FUNCTION_BLOCK numeroDePartidas (* Basic Function Block Type *)
  (* Standard: 61499-2 *)
  (* Version 0.0, 14/01/2026, Schneider Electric, Template *)
  PACKAGE Hidryco.HidrycoLib;
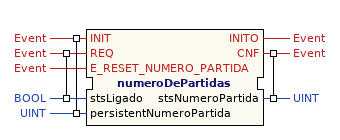
  EVENT_INPUT
    INIT WITH persistentNumeroPartida; (* Initialization Request *)
    REQ WITH stsLigado; (* Normal Execution Request *)
    E_RESET_NUMERO_PARTIDA;
  END_EVENT
  EVENT_OUTPUT
    INITO; (* Initialization Confirm *)
    CNF WITH stsNumeroPartida; (* Execution Confirmation *)
  END_EVENT
  VAR_INPUT
    stsLigado : BOOL;
    persistentNumeroPartida : UINT;
  END_VAR
  VAR_OUTPUT
    stsNumeroPartida : UINT; (* Output event qualifier *)
  END_VAR
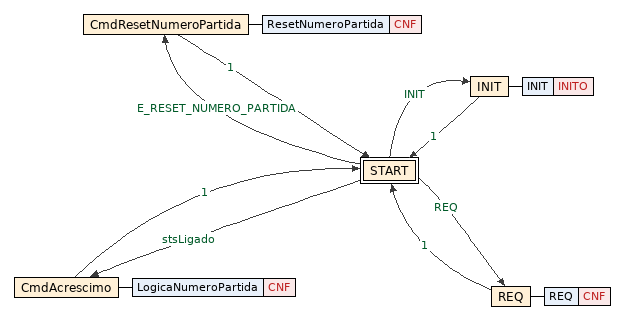
  EC_STATES
    START; (* Initial State *)
    INIT : INIT -> INITO; (* Initialization *)
    REQ : REQ -> CNF; (* Normal execution *)
    CmdAcrescimo : LogicaNumeroPartida -> CNF;
    CmdResetNumeroPartida : ResetNumeroPartida -> CNF;
  END_STATES
  EC_TRANSITIONS
    START TO INIT := INIT;
    INIT TO START := 1;
    START TO REQ := REQ;
    REQ TO START := 1;
    START TO CmdAcrescimo := stsLigado;
    CmdAcrescimo TO START := 1;
    START TO CmdResetNumeroPartida := E_RESET_NUMERO_PARTIDA;
    CmdResetNumeroPartida TO START := 1;
  END_TRANSITIONS
  ALGORITHM INIT IN ST: (* Initialization algorithm *)
stsNumeroPartida := persistentNumeroPartida;
;
  END_ALGORITHM
  ALGORITHM REQ IN ST: (* Normally executed algorithm *)
;
  END_ALGORITHM
  ALGORITHM LogicaNumeroPartida IN ST:
stsNumeroPartida := stsNumeroPartida + 1;
;
  END_ALGORITHM
  ALGORITHM ResetNumeroPartida IN ST:
stsNumeroPartida  := 0;
;
  END_ALGORITHM
END_FUNCTION_BLOCK
